// TwinCAT 3 PLC project demo_pcl_vm
// ProgramVersion: 3.1.4024.0
// libraries:
//   Tc2_Standard, * (Beckhoff Automation GmbH)
//   Tc2_System, * (Beckhoff Automation GmbH)
//   Tc3_Module, * (Beckhoff Automation GmbH)
//   VisuSymbols,3.5.10.0,System
// project tree:
//   / GlobalTextList.TcGTLO, PlcTask.TcTTO, Visualization Manager.TcVMO (not stored), Visualization.TcVIS
//   GVLs/ GVL.TcGVL
//   POUs/ MAIN.TcPOU

CONFIGURATION demo_pcl_vm
    RESOURCE PLC ON TwinCAT3
        TASK PlcTask(INTERVAL := T#10ms, PRIORITY := 20);
        PROGRAM MAIN WITH PlcTask : MAIN;
    END_RESOURCE
END_CONFIGURATION

// ---- GVLs/GVL.TcGVL
{attribute 'qualified_only'}
VAR_GLOBAL
	button_pressed : BOOL;
	lamp_on : BOOL;
END_VAR

// ---- POUs/MAIN.TcPOU
PROGRAM MAIN
VAR
	my_counter : INT := 0;
	btn : BOOL;
	lmp : BOOL;
END_VAR

my_counter := my_counter + 2;

gvl.lamp_on := gvl.button_pressed;

END_PROGRAM

// ---- Visualization.TcVIS
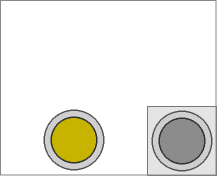
VISUALIZATION Visualization  // 217x176
    Lamp1 (39,105 70x70), variable: GVL.lamp_on, style: Lamp-Lamp1-Yellow
    PushSwitch (147,106 70x70), variable: GVL.button_pressed, behaviour: TOGGLE, style: Switch-PushSwitch-Gray
END_VISUALIZATION
